{attribute 'qualified_only'}
{attribute 'strict'}
TYPE BarcodeVerificationResult :
(
	UNVERIFIED 	:= 0,
	VALID		:= 1,
	INVALID		:= 2
);
END_TYPE

(* stored: Version 1.1.0.1, ProductVersion 3.1.4024.12
   DUT BarcodeVerificationResult: Id {4113fdb6-8cca-484a-a578-3356ae40acec} *)
